(*

.. <legal notes>

legal notes
=================
| SPDX-FileCopyrightText: © 2026 Oleksandr Tiutyk <trofimich@gmail.com>
| SPDX-License-Identifier: LGPL-3.0-only
| For details check: LGPL-3.0-only_

.. _LGPL-3.0-only: https://www.gnu.org/licenses/lgpl-3.0.en.html

.. </legal notes>

*)

{attribute 'qualified_only'}
{attribute 'strict'}
{attribute 'to_string'}
TYPE TRAFFIC_LIGHT_COLOR :
(
	NO_COLOR := 0,
	RED,
	YELLOW,
	GREEN
);
END_TYPE

(* stored: Version 1.1.0.1
   DUT TRAFFIC_LIGHT_COLOR: Id {773330fa-d0f3-4bdf-bce6-a9f585e1025a} *)
